// SIMATIC S7-200 project (STEP 7-Micro/WIN), CPU 224 REL 02.00

SYMBOL_TABLE 用户1
自动/手动开关          I0.0
秤放料按钮2           M0.0
放成品按钮2           M0.1
搅拌器按钮2           M0.2
进1号料按钮2          M0.3
进2号料按钮2          M0.4
进3号料按钮2          M0.5
进4号料按钮2          M0.6
起动按钮2            M0.7
停止按钮2            M1.0
进4号料阀            Q1.0
秤放料阀             Q0.2
放成品阀             Q0.3
搅拌电动机            Q0.4
进1号料阀            Q0.5
进2号料阀            Q0.6
进3号料阀            Q0.7
搅拌转速测量值          VW10
1号料当前重量          VW12
2号料当前重量          VW14
3号料当前重量          VW16
4号料当前重量          VW18
事故信息             VW2
1号料累加值           VW20
2号料累加值           VW22
3号料累加值           VW24
4号料累加值           VW26
秤斗料位             VW42
混合仓料位            VW44
皮重               VW46
总重量              VW60
IW替代值            VW62
秤放料时间            VW64
搅拌时间             VW66
放成品时间            VW68
配方编号             VW6
读配方              M1.1
写配方              M1.2
END_SYMBOL_TABLE

ORGANIZATION_BLOCK 主:OB1
TITLE=程序注解
BEGIN
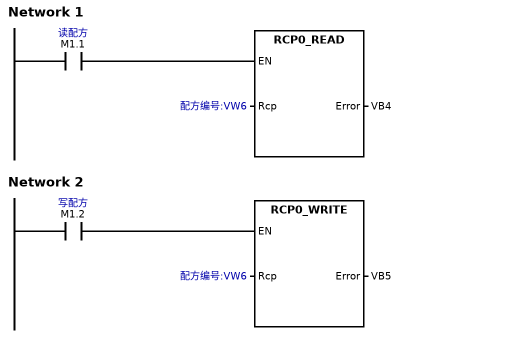
Network 1
LD     读配方:M1.1
CALL   RCP0_READ:SBR1, 配方编号:VW6, VB4
Network 2
LD     写配方:M1.2
CALL   RCP0_WRITE:SBR2, 配方编号:VW6, VB5
END_ORGANIZATION_BLOCK

// SBR1: protected block, not included

// SBR2: protected block, not included

// (further data pages could not be read)
